{attribute 'qualified_only'}
VAR_GLOBAL
	Control : TYP_PRES_CNTRL_CONTROL;
	Parameter : TYP_PRES_CNTRL_PARAMETER;
	Status : TYP_PRES_CNTRL_STATUS;
END_VAR

(* stored: Version 1.1.0.1, ProductVersion 3.1.4024.12
   GVL gPresCntrl: Id {552cff3f-2caa-4ec0-ae22-28f9457d3769} *)
